// TIA Portal V17 export
// export: Created 2023-12-22T15:03:17.7573407Z, ExportSetting WithDefaults, DisplayName Totally Integrated Automation Portal, DisplayVersion V17, DisplayName TIA Portal Openness, DisplayVersion V17, DisplayName TIA Portal Version Control Interface, DisplayVersion V17, DisplayName STEP 7 Professional, DisplayVersion V17, DisplayName STEP 7 Safety, DisplayVersion V17, DisplayName WinCC Advanced, DisplayVersion V17
DATA_BLOCK "SKV_Main_DB"   // DB15
VERSION : 0.1
// stored: AutoNumber true, DBAccessibleFromOPCUA true, DBAccessibleFromWebserver true, InstanceOfName SKV_Main, InstanceOfType FB
"SKV_Main"
   // VAR RETAIN
   //    One { S7_SetPoint := 'True'} : Array[0..11] of "SKV_One";
   //    SP : Struct
   //       Max { S7_SetPoint := 'True'} : Real := 0.0;
   //       High : Real;
   //       Auto : Real;
   //       Point : Real;
   //       Low : Real;
   //       Min { S7_SetPoint := 'True'} : Real := 0.0;
   //    END_STRUCT;
   //    cnt : Struct
   //       Min { S7_SetPoint := 'True'} : Int := 0;
   //       Fix { S7_SetPoint := 'True'} : Int := 2;
   //       All : Int;
   //       Group : Int;
   //       Reserve : Int;
   //       Ready : Int;
   //       Low : Int;
   //       Work : Int;
   //       Start : Int;
   //    END_STRUCT;
   //    tmp : Int;
   // END_VAR
BEGIN
   One[0..11].SP_Use := TRUE;
   One[0].Mode := 0;
   One[1..11].Mode := 1;
   One[0..11].C := 0.0;
   One[0..11].SP.Low_Percent := 85.0;
   One[0..11].SP.Min := 30.0;
   One[0..11].SP.Max := 45.0;
   One[0..11].SP.Delta := 10.0;
END_DATA_BLOCK
